{attribute addProperty BoxType "EP2001-1000-0016"}
{attribute addProperty Id "Output1AT %Q*BOOL811Output2AT %Q*BOOL812Output3AT %Q*BOOL813Output4AT %Q*BOOL814"}
{attribute addProperty CRC "1411626247"}
{attribute addProperty SizeInBites "32"}
{attribute addProperty SizeInBytes "4"}
TYPE Group_5423B507 :
STRUCT
	{attribute addProperty Name "Output1"}
	Output1 AT %Q* : BOOL;
	{attribute addProperty Name "Output2"}
	Output2 AT %Q* : BOOL;
	{attribute addProperty Name "Output3"}
	Output3 AT %Q* : BOOL;
	{attribute addProperty Name "Output4"}
	Output4 AT %Q* : BOOL;
END_STRUCT
END_TYPE

(* stored: Version 1.2.0.0, ProductVersion 3.1.4024.9
   DUT Group_5423B507: Id {f5cc448b-119f-45f5-94cc-c52321778090} *)
